PROGRAM PRG_LARS_02_GateSeparationCtrl
VAR
	fbPerformance						: FB_Interval;

	tonGateReleaseNoPrint		: TON;
	tonGateReleaseTimeOut	: TON;
	bRelaesGateActive		: BOOL;
	tonGateClose	: TON;

	rsClamptState		: RS;
	rsGateState		: RS;

	ftrigLabelPrinted		: F_TRIG;
	rtrigAplicatorAtHome	: R_TRIG;
	bFastRelease			: BOOL;
END_VAR
VAR // added by the converter: edge detectors and wires of the graphical bodies
    _w1 : BOOL;
END_VAR

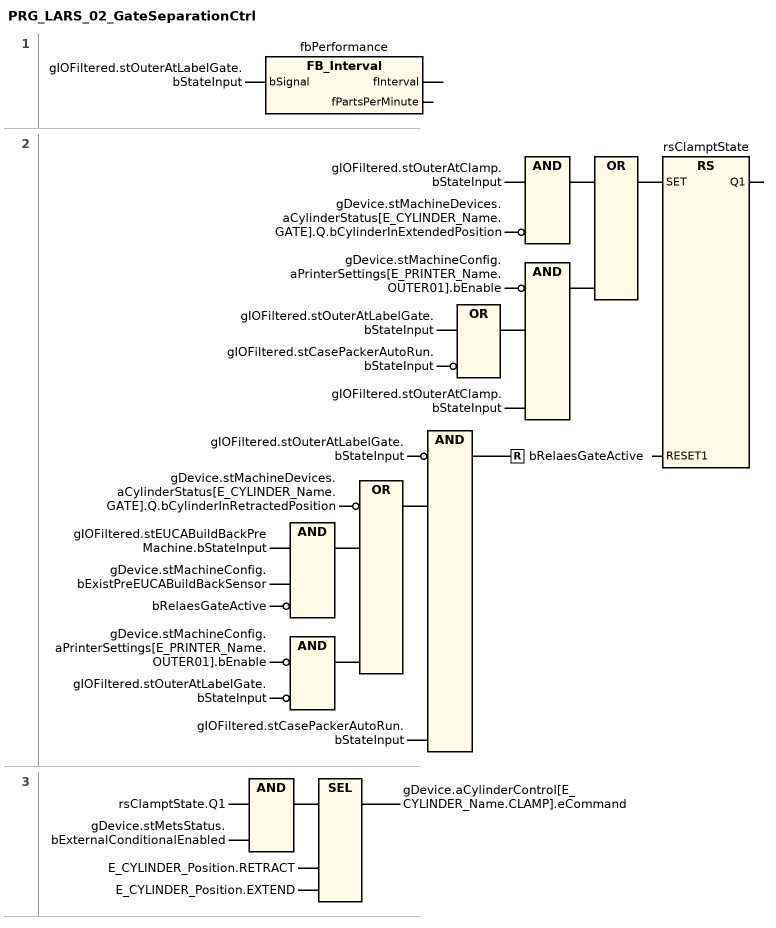
// NETWORK 1
fbPerformance(bSignal := gIOFiltered.stOuterAtLabelGate.bStateInput); // FB_Interval

// NETWORK 2
_w1 := NOT gIOFiltered.stOuterAtLabelGate.bStateInput AND (NOT gDevice.stMachineDevices.aCylinderStatus[E_CYLINDER_Name.GATE].Q.bCylinderInRetractedPosition OR gIOFiltered.stEUCABuildBackPreMachine.bStateInput AND gDevice.stMachineConfig.bExistPreEUCABuildBackSensor AND NOT bRelaesGateActive OR NOT gDevice.stMachineConfig.aPrinterSettings[E_PRINTER_Name.OUTER01].bEnable AND NOT gIOFiltered.stOuterAtLabelGate.bStateInput) AND gIOFiltered.stCasePackerAutoRun.bStateInput;
bRelaesGateActive R= _w1;
rsClamptState(SET := gIOFiltered.stOuterAtClamp.bStateInput AND NOT gDevice.stMachineDevices.aCylinderStatus[E_CYLINDER_Name.GATE].Q.bCylinderInExtendedPosition OR NOT gDevice.stMachineConfig.aPrinterSettings[E_PRINTER_Name.OUTER01].bEnable AND (gIOFiltered.stOuterAtLabelGate.bStateInput OR NOT gIOFiltered.stCasePackerAutoRun.bStateInput) AND gIOFiltered.stOuterAtClamp.bStateInput, RESET1 := _w1); // RS

// NETWORK 3
gDevice.aCylinderControl[E_CYLINDER_Name.CLAMP].eCommand := SEL(rsClamptState.Q1 AND gDevice.stMetsStatus.bExternalConditionalEnabled, E_CYLINDER_Position.RETRACT, E_CYLINDER_Position.EXTEND);

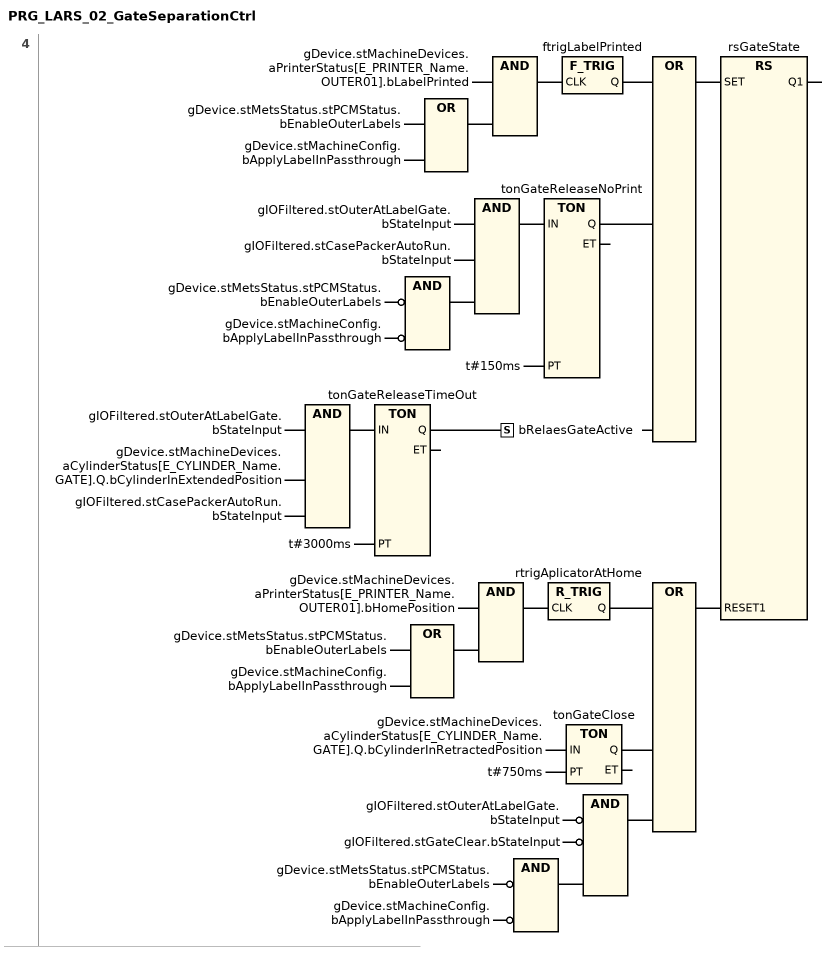
// NETWORK 4
ftrigLabelPrinted(CLK := gDevice.stMachineDevices.aPrinterStatus[E_PRINTER_Name.OUTER01].bLabelPrinted AND (gDevice.stMetsStatus.stPCMStatus.bEnableOuterLabels OR gDevice.stMachineConfig.bApplyLabelInPassthrough)); // F_TRIG
tonGateReleaseNoPrint(IN := gIOFiltered.stOuterAtLabelGate.bStateInput AND gIOFiltered.stCasePackerAutoRun.bStateInput AND (NOT gDevice.stMetsStatus.stPCMStatus.bEnableOuterLabels AND NOT gDevice.stMachineConfig.bApplyLabelInPassthrough), PT := t#150ms); // TON
tonGateReleaseTimeOut(IN := gIOFiltered.stOuterAtLabelGate.bStateInput AND gDevice.stMachineDevices.aCylinderStatus[E_CYLINDER_Name.GATE].Q.bCylinderInExtendedPosition AND gIOFiltered.stCasePackerAutoRun.bStateInput, PT := t#3000ms); // TON
bRelaesGateActive S= tonGateReleaseTimeOut.Q;
rtrigAplicatorAtHome(CLK := gDevice.stMachineDevices.aPrinterStatus[E_PRINTER_Name.OUTER01].bHomePosition AND (gDevice.stMetsStatus.stPCMStatus.bEnableOuterLabels OR gDevice.stMachineConfig.bApplyLabelInPassthrough)); // R_TRIG
tonGateClose(IN := gDevice.stMachineDevices.aCylinderStatus[E_CYLINDER_Name.GATE].Q.bCylinderInRetractedPosition, PT := t#750ms); // TON
rsGateState(SET := ftrigLabelPrinted.Q OR tonGateReleaseNoPrint.Q OR tonGateReleaseTimeOut.Q, RESET1 := rtrigAplicatorAtHome.Q OR tonGateClose.Q OR NOT gIOFiltered.stOuterAtLabelGate.bStateInput AND NOT gIOFiltered.stGateClear.bStateInput AND (NOT gDevice.stMetsStatus.stPCMStatus.bEnableOuterLabels AND NOT gDevice.stMachineConfig.bApplyLabelInPassthrough)); // RS

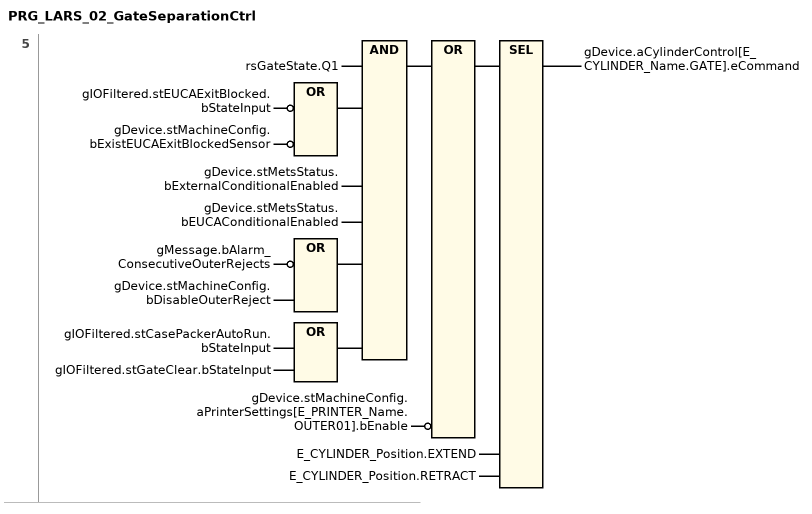
// NETWORK 5
gDevice.aCylinderControl[E_CYLINDER_Name.GATE].eCommand := SEL(rsGateState.Q1 AND (NOT gIOFiltered.stEUCAExitBlocked.bStateInput OR NOT gDevice.stMachineConfig.bExistEUCAExitBlockedSensor) AND gDevice.stMetsStatus.bExternalConditionalEnabled AND gDevice.stMetsStatus.bEUCAConditionalEnabled AND (NOT gMessage.bAlarm_ConsecutiveOuterRejects OR gDevice.stMachineConfig.bDisableOuterReject) AND (gIOFiltered.stCasePackerAutoRun.bStateInput OR gIOFiltered.stGateClear.bStateInput) OR NOT gDevice.stMachineConfig.aPrinterSettings[E_PRINTER_Name.OUTER01].bEnable, E_CYLINDER_Position.EXTEND, E_CYLINDER_Position.RETRACT);

END_PROGRAM

(* stored: Version 1.1.0.1
   POU PRG_LARS_02_GateSeparationCtrl: Id {381a740f-ed8f-463e-a946-0104463fa9c0}, SpecialFunc None *)
